(* IEC 61131-3 sources: elevator-digital-twin/codesys, 11 files *)

(* ---- DUT_Types.st ---- *)
(*
    ============================================================================
    DUT_Types.st   —   Asansor Digital Twin / Veri tipleri
    CODESYS 3.5 SP17+  |  Structured Text
    ----------------------------------------------------------------------------
    NOT: Bu dosyadaki her TYPE blogu, CODESYS projesinde AYRI bir DUT nesnesi
         olarak olusturulmalidir (Application > Add Object > DUT).
    NOT: Buradaki sayisal degerler Godot tarafinda scripts/IoMap.gd ve
         scripts/Config.gd icinde birebir ayni tanimlanmistir. Birini
         degistirirseniz digerini de degistirin.
    ============================================================================
*)

// ---------------------------------------------------------------------------
// Ana durum makinesi durumlari  (Godot: IoMap.State)
// ---------------------------------------------------------------------------
TYPE E_LiftState :
(
    LS_INIT         := 0,   // guc geldi, henuz konum bilinmiyor
    LS_HOMING       := 1,   // referans kata inis
    LS_IDLE         := 2,   // bosta, cagri bekliyor
    LS_DOOR_OPENING := 3,
    LS_DOOR_OPEN    := 4,   // bekleme suresi (dwell) sayiyor
    LS_DOOR_CLOSING := 5,
    LS_START        := 6,   // fren cozme + surucu enable
    LS_TRAVEL       := 7,   // nominal hizda seyir
    LS_DECEL        := 8,   // yavaslama rampasi
    LS_LEVEL        := 9,   // kat seviyeleme (surunme hizi)
    LS_ARRIVED      := 10,  // durdu, fren tuttu
    LS_FAULT        := 11,
    LS_FIRE         := 12,  // yangin senaryosu
    LS_INSPECTION   := 13,  // revizyon (kabin ustu kumanda)
    LS_PARK         := 14   // park katina donus
) INT;
END_TYPE

// ---------------------------------------------------------------------------
// Yon  (Godot: IoMap.DIR_*)
// ---------------------------------------------------------------------------
TYPE E_Direction :
(
    DIR_NONE := 0,
    DIR_UP   := 1,
    DIR_DOWN := 2
) INT;
END_TYPE

// ---------------------------------------------------------------------------
// Kapi alt durum makinesi
// ---------------------------------------------------------------------------
TYPE E_DoorState :
(
    DS_CLOSED  := 0,
    DS_OPENING := 1,
    DS_OPEN    := 2,
    DS_CLOSING := 3,
    DS_REOPEN  := 4,   // foto bariyer kesildi, geri ac
    DS_FAULT   := 5
) INT;
END_TYPE

// ---------------------------------------------------------------------------
// Hata kodlari  (Godot: IoMap.FAULT_TEXT)
// ---------------------------------------------------------------------------
TYPE E_Fault :
(
    FLT_NONE          := 0,
    FLT_SAFETY_CHAIN  := 1,   // guvenlik devresi acik
    FLT_DOOR_TIMEOUT  := 2,   // kapi verilen surede kapanmadi/acilmadi
    FLT_TRAVEL_TIMEOUT:= 3,   // kat arasi sure asildi
    FLT_DRIVE         := 4,   // surucu hazir degil / surucu arizasi
    FLT_LIMIT         := 5,   // ucdaki limit switch'e carpildi
    FLT_ENCODER       := 6,   // encoder ile kat sensoru uyusmuyor
    FLT_LOCK_LOST     := 7,   // hareket sirasinda kapi kilidi acildi
    FLT_ESTOP         := 8,   // acil stop butonu
    FLT_BRAKE         := 9,   // fren geri beslemesi kumandayla uyusmuyor
    FLT_OVERSPEED     := 10   // hiz regulatoru devreye girdi
) INT;
END_TYPE

// ---------------------------------------------------------------------------
// Cagri kayit kumesi — dispatcher bu yapinin uzerinde calisir
// ---------------------------------------------------------------------------
TYPE ST_CallSet :
STRUCT
    axUp   : ARRAY[0..15] OF BOOL;   // kat holu YUKARI cagrilari
    axDown : ARRAY[0..15] OF BOOL;   // kat holu ASAGI cagrilari
    axCar  : ARRAY[0..15] OF BOOL;   // kabin ici kat butonlari
END_STRUCT
END_TYPE

// ---------------------------------------------------------------------------
// Sahadan gelen sinyaller  (Godot fizik modeli uretir -> Modbus -> buraya)
// ---------------------------------------------------------------------------
TYPE ST_LiftInputs :
STRUCT
    // Butonlar (momentary)
    stCalls        : ST_CallSet;
    xDoorOpenBtn   : BOOL;
    xDoorCloseBtn  : BOOL;
    xAlarmBtn      : BOOL;
    xFaultReset    : BOOL;

    // Kuyu / kabin sensorleri
    axFloorZone    : ARRAY[0..15] OF BOOL;  // kat seviye (door zone) bayragi
    diPosMM        : DINT;                  // mutlak encoder konumu [mm]
    iActSpeedMMS   : INT;                   // gercek hiz [mm/s]
    iDoorPosPmil   : INT;                   // kapi konumu 0..1000 (0=kapali)
    iLoadKg        : INT;

    // Guvenlik zinciri ve limitler
    xTopLimit      : BOOL;
    xBotLimit      : BOOL;
    xDoorOpenLimit : BOOL;
    xDoorCloseLimit: BOOL;
    xDoorLocked    : BOOL;   // kat kapisi kilit kontagi zinciri
    xBrakeFb       : BOOL;   // fren geri bildirimi
    xSafetyChain   : BOOL;   // TRUE = zincir saglam
    xGovernorOk    : BOOL;   // hiz regulatoru saglam

    // Mod secicileri
    xEStop         : BOOL;
    xOverload      : BOOL;
    xObstruction   : BOOL;   // foto bariyer kesildi
    xFireCall      : BOOL;
    xInspection    : BOOL;
    xInspUp        : BOOL;
    xInspDown      : BOOL;
    xDriveReady    : BOOL;
    xDriveFault    : BOOL;
END_STRUCT
END_TYPE

// ---------------------------------------------------------------------------
// PLC cikislari  (Modbus -> Godot fizik modeli + gorsel)
// ---------------------------------------------------------------------------
TYPE ST_LiftOutputs :
STRUCT
    // Surucu
    xDriveEnable  : BOOL;
    xRunUp        : BOOL;
    xRunDown      : BOOL;
    xBrakeRelease : BOOL;
    xLeveling     : BOOL;
    iSpeedSpMMS   : INT;

    // Kapi
    xDoorOpen     : BOOL;
    xDoorClose    : BOOL;
    xDoorNudge    : BOOL;   // yavas zorlamali kapama

    // Lambalar
    axLampUp      : ARRAY[0..15] OF BOOL;
    axLampDown    : ARRAY[0..15] OF BOOL;
    axLampCar     : ARRAY[0..15] OF BOOL;

    // Gosterge / durum
    iCurrentFloor : INT;
    iTargetFloor  : INT;
    eDirection    : E_Direction;
    eState        : E_LiftState;
    eFault        : E_Fault;
    xMoving       : BOOL;
    xDoorIsOpen   : BOOL;
    xDoorIsClosed : BOOL;
    xOverloadLamp : BOOL;
    xFaultLamp    : BOOL;
    xFireMode     : BOOL;
    xInspMode     : BOOL;
    xOutOfService : BOOL;
    xGong         : BOOL;
    xAlarm        : BOOL;   // alarm zili (kabin alarm butonu)
    xCabinLight   : BOOL;
    iDoorTimerMs  : INT;    // kalan bekleme suresi [ms]
    iHeartbeat    : INT;
END_STRUCT
END_TYPE

(* ---- GVL_Config.st ---- *)
(*
    ============================================================================
    GVL_Config   —   Tesis parametreleri (tek kaynak)
    Application > Add Object > Global Variable List  adiyla: GVL_Config
    ----------------------------------------------------------------------------
    !! Godot tarafindaki karsiligi: godot/scripts/Config.gd
       Iki dosyadaki degerler ayni olmak zorunda, yoksa twin ile gercek PLC
       farkli davranir.
    ============================================================================
*)
VAR_GLOBAL CONSTANT

    // --- Kuyu geometrisi ----------------------------------------------------
    C_FLOOR_COUNT      : INT  := 6;      // 0 = zemin ... 5 = en ust kat
    C_TOP_FLOOR        : INT  := 5;
    C_FLOOR_HEIGHT_MM  : DINT := 3200;   // katlar arasi mesafe
    C_DOOR_ZONE_MM     : DINT := 60;     // kat seviyesi +/- door-zone bolgesi
    C_LEVEL_TOL_MM     : DINT := 8;      // "kata geldi" toleransi
    C_OVERTRAVEL_MM    : DINT := 400;    // ucdaki limit switch mesafesi

    // --- Surus profili ------------------------------------------------------
    C_V_RATED_MMS      : INT  := 1600;   // nominal hiz
    C_V_LEVEL_MMS      : INT  := 150;    // seviyeleme (surunme) hizi
    C_V_INSPECT_MMS    : INT  := 300;    // revizyon hizi
    C_V_OVERSPEED_MMS  : INT  := 1840;   // regulator devreye girme hizi (%115)
    C_DECEL_DIST_MM    : DINT := 2000;   // yavaslamaya baslama mesafesi
                                         // (jerk sinirli surucunun durma
                                         //  mesafesine gore boyutlandirildi)

    // --- Zamanlar -----------------------------------------------------------
    C_T_DOOR_DWELL     : TIME := T#4S;    // kabin cagrisinda kapi acik kalma
    C_T_DOOR_DWELL_HALL: TIME := T#3S;    // sadece hol cagrisinda
    C_T_DOOR_MOVE_MAX  : TIME := T#8S;    // kapi hareket zaman asimi
    C_T_TRAVEL_MAX     : TIME := T#25S;   // kat arasi hareket zaman asimi
    C_T_NUDGE          : TIME := T#15S;   // bu sureden sonra zorlamali kapama
    C_T_GONG           : TIME := T#600MS;
    C_T_PARK           : TIME := T#30S;   // bosta bekleyince park katina don
    C_T_BRAKE          : TIME := T#300MS; // fren cozme/tutma gecikmesi
    C_T_START_DELAY    : TIME := T#200MS; // surucu enable -> hareket
    C_T_ALARM          : TIME := T#2S;    // alarm zili calma suresi
    C_T_BRAKE_FB       : TIME := T#1S;    // fren geri besleme denetimi
    C_T_OVERSPEED      : TIME := T#300MS; // asiri hiz onaylama suresi

    // --- Kat / yuk ----------------------------------------------------------
    C_PARK_FLOOR       : INT  := 0;
    C_FIRE_FLOOR       : INT  := 0;      // yangin tahliye kati
    C_LOAD_FULL_KG     : INT  := 630;
    C_LOAD_OVER_KG     : INT  := 693;    // %110 -> asiri yuk

END_VAR

(* ---- GVL_IO.st ---- *)
(*
    ============================================================================
    GVL_IO   —   Modbus TCP Slave Device register alani
    Application > Add Object > Global Variable List  adiyla: GVL_IO
    ----------------------------------------------------------------------------
    CODESYS "Modbus TCP Slave Device" mantigi:
       Holding Registers  -> PLC girisi  (%IW)  : Godot yazar, PLC okur
       Input Registers    -> PLC cikisi  (%QW)  : PLC yazar, Godot okur

    ONEMLI: Asagidaki %IW0 / %QW0 baslangic adresleri sizin projenizde farkli
    olabilir. Cihaz agacinda "Modbus_TCP_Slave_Device > Modbus TCP Slave Device
    I/O Mapping" sekmesini acip gercek baslangic adresini gorun ve buradaki
    AT ifadelerini ona gore duzeltin.

    Alternatif (AT kullanmak istemezseniz): AT ifadelerini silin, dizileri
    normal degisken birakin ve I/O Mapping sekmesinde her kanali tek tek
    GVL_IO.g_awMbIn[x] / g_awMbOut[x] degiskenine baglayin.
    ============================================================================
*)
VAR_GLOBAL

    // Godot -> PLC  (Holding Registers, master write)
    g_awMbIn  AT %IW0 : ARRAY[0..15] OF WORD;

    // PLC -> Godot  (Input Registers, master read)
    g_awMbOut AT %QW0 : ARRAY[0..15] OF WORD;

    // Uygulama katmani (PRG_ModbusIO tarafindan doldurulur / okunur)
    g_stIn  : ST_LiftInputs;
    g_stOut : ST_LiftOutputs;

    // Baglanti gozetimi
    g_xTwinOnline   : BOOL;        // Godot heartbeat degisiyor mu
    g_iTwinHbLast   : INT;
    g_tTwinLostTime : TIME;

END_VAR

(*
    ============================================================================
    REGISTER HARITASI  (docs/io-map.md ile ayni)
    ----------------------------------------------------------------------------
    Godot -> PLC   g_awMbIn[n]    (Holding Register n)
      0  HALL_UP        bit n = n. kat YUKARI cagri butonu
      1  HALL_DOWN      bit n = n. kat ASAGI cagri butonu
      2  CAR_CALL       bit n = kabin ici n. kat butonu
      3  CMD_BITS       0 kapi-ac btn      1 kapi-kapa btn   2 alarm
                        3 acil stop        4 asiri yuk       5 yangin cagrisi
                        6 revizyon         7 hata reset      8 foto bariyer
                        9 surucu hazir    10 surucu ariza   11 revizyon YUKARI
                       12 revizyon ASAGI
      4  FLOOR_ZONE     bit n = kabin n. katin door-zone bolgesinde
      5  LIMIT_BITS     0 ust limit        1 alt limit       2 kapi acik limit
                        3 kapi kapali lim. 4 kapi kilidi     5 fren geri bes.
                        6 guvenlik zinciri 7 hiz regulatoru
      6  CAR_POS_MM     mutlak konum [mm]  (0..65535)
      7  CAR_SPEED_MMS  gercek hiz [mm/s]
      8  DOOR_POS_PMIL  kapi konumu 0..1000
      9  LOAD_KG        kabin yuku [kg]
     10  TWIN_HB        Godot heartbeat (her cevrim +1)
     11..15  rezerve

    PLC -> Godot   g_awMbOut[n]   (Input Register n)
      0  DRIVE_CMD      0 enable  1 yukari  2 asagi  3 fren-coz  4 seviyeleme
      1  DOOR_CMD       0 ac      1 kapa    2 nudge
      2  LAMP_HALL_UP   bit n
      3  LAMP_HALL_DOWN bit n
      4  LAMP_CAR       bit n
      5  STATUS_BITS    0 hareket  1 kapi acik  2 kapi kapali  3 asiri yuk
                        4 ariza    5 yangin     6 revizyon     7 servis disi
                        8 gong     9 ok-yukari 10 ok-asagi    11 kabin lambasi
                       12 alarm zili
      6  CURRENT_FLOOR
      7  TARGET_FLOOR
      8  DIRECTION      0 yok 1 yukari 2 asagi
      9  SPEED_SP_MMS   hiz referansi [mm/s]
     10  STATE_CODE     E_LiftState
     11  FAULT_CODE     E_Fault
     12  PLC_HB         PLC heartbeat
     13  DOOR_TIMER_MS  kapi bekleme kalan sure [ms]
     14..15  rezerve
    ============================================================================
*)

(* ---- FUN_Bits.st ---- *)
(*
    ============================================================================
    Bit yardimci fonksiyonlari
    Her FUNCTION ayri bir POU olarak eklenmelidir (Add Object > POU > Function).
    ============================================================================
*)

FUNCTION F_GetBit : BOOL
VAR_INPUT
    wVal : WORD;
    iBit : INT;
END_VAR

IF (iBit < 0) OR (iBit > 15) THEN
    F_GetBit := FALSE;
ELSE
    F_GetBit := (wVal AND SHL(WORD#1, INT_TO_BYTE(iBit))) <> 0;
END_IF

END_FUNCTION

FUNCTION F_SetBit : WORD
VAR_INPUT
    wVal : WORD;
    iBit : INT;
    xVal : BOOL;
END_VAR

IF (iBit < 0) OR (iBit > 15) THEN
    F_SetBit := wVal;
ELSIF xVal THEN
    F_SetBit := wVal OR SHL(WORD#1, INT_TO_BYTE(iBit));
ELSE
    F_SetBit := wVal AND (NOT SHL(WORD#1, INT_TO_BYTE(iBit)));
END_IF

END_FUNCTION

(* ---- FB_CallRegistry.st ---- *)
(*
    ============================================================================
    FB_CallRegistry   —   Cagri kaydi (latch) ve lamba surme
    ----------------------------------------------------------------------------
    Butonlar momentary gelir; bu blok cagriyi tutar, servis edilince siler.
    Godot karsiligi: SoftPlc.gd -> class CallRegistry
    ============================================================================
*)
FUNCTION_BLOCK FB_CallRegistry
VAR_INPUT
    stBtn       : ST_CallSet;     // sahadan gelen anlik buton durumu
    xClearAll   : BOOL;           // yangin / revizyon / ariza -> tum cagrilari sil
    xEnable     : BOOL;           // FALSE ise yeni cagri kabul etme
END_VAR
VAR_IN_OUT
    stLatch     : ST_CallSet;     // kalici cagri kaydi (dispatcher ile paylasilir)
END_VAR
VAR_OUTPUT
    xAnyCall    : BOOL;
    iCallCount  : INT;
END_VAR
VAR
    i : INT;
END_VAR

// ---------------------------------------------------------------------------
IF xClearAll THEN
    FOR i := 0 TO 15 DO
        stLatch.axUp[i]   := FALSE;
        stLatch.axDown[i] := FALSE;
        stLatch.axCar[i]  := FALSE;
    END_FOR
    xAnyCall   := FALSE;
    iCallCount := 0;
    RETURN;
END_IF

xAnyCall   := FALSE;
iCallCount := 0;

FOR i := 0 TO C_TOP_FLOOR DO

    // --- yeni cagrilari yakala -------------------------------------------
    IF xEnable THEN
        // en ust katta yukari, en alt katta asagi butonu yoktur
        IF stBtn.axUp[i]   AND (i < C_TOP_FLOOR) THEN stLatch.axUp[i]   := TRUE; END_IF
        IF stBtn.axDown[i] AND (i > 0)           THEN stLatch.axDown[i] := TRUE; END_IF
        IF stBtn.axCar[i]                        THEN stLatch.axCar[i]  := TRUE; END_IF
    END_IF

    // --- sayim -------------------------------------------------------------
    IF stLatch.axUp[i]   THEN iCallCount := iCallCount + 1; END_IF
    IF stLatch.axDown[i] THEN iCallCount := iCallCount + 1; END_IF
    IF stLatch.axCar[i]  THEN iCallCount := iCallCount + 1; END_IF

END_FOR

xAnyCall := (iCallCount > 0);

(*
    ---------------------------------------------------------------------------
    METHOD ServeFloor : Bir katta durulduğunda o kata ait cagrilari siler.
    eDir = hangi yonun cagrisi servis edildi (DIR_NONE ise ikisi de silinir)
    ---------------------------------------------------------------------------
*)
METHOD ServeFloor
VAR_INPUT
    iFloor : INT;
    eDir   : E_Direction;
END_VAR

IF (iFloor < 0) OR (iFloor > C_TOP_FLOOR) THEN RETURN; END_IF

stLatch.axCar[iFloor] := FALSE;

CASE eDir OF
    DIR_UP:
        stLatch.axUp[iFloor] := FALSE;
        // ileride cagri kalmadiysa ters yon cagrisini da al
        IF NOT THIS^.CallAbove(iFloor) THEN
            stLatch.axDown[iFloor] := FALSE;
        END_IF

    DIR_DOWN:
        stLatch.axDown[iFloor] := FALSE;
        IF NOT THIS^.CallBelow(iFloor) THEN
            stLatch.axUp[iFloor] := FALSE;
        END_IF
ELSE
    stLatch.axUp[iFloor]   := FALSE;
    stLatch.axDown[iFloor] := FALSE;
END_CASE

END_METHOD

(*  Verilen katin USTUNDE bekleyen herhangi bir cagri var mi?  *)
METHOD CallAbove : BOOL
VAR_INPUT
    iFloor : INT;
END_VAR
VAR
    k : INT;
END_VAR

CallAbove := FALSE;
FOR k := iFloor + 1 TO C_TOP_FLOOR DO
    IF stLatch.axUp[k] OR stLatch.axDown[k] OR stLatch.axCar[k] THEN
        CallAbove := TRUE;
        RETURN;
    END_IF
END_FOR

END_METHOD

(*  Verilen katin ALTINDA bekleyen herhangi bir cagri var mi?  *)
METHOD CallBelow : BOOL
VAR_INPUT
    iFloor : INT;
END_VAR
VAR
    k : INT;
END_VAR

CallBelow := FALSE;
FOR k := 0 TO iFloor - 1 DO
    IF stLatch.axUp[k] OR stLatch.axDown[k] OR stLatch.axCar[k] THEN
        CallBelow := TRUE;
        RETURN;
    END_IF
END_FOR

END_METHOD

(* ---- FB_Dispatcher.st ---- *)
(*
    ============================================================================
    FB_Dispatcher   —   Hedef kat secimi  (collective control / toplamali kumanda)
    ----------------------------------------------------------------------------
    Kural:
      * Kabin bir yone gidiyorsa o yondeki tum cagrilari sirasiyla toplar.
      * Yonunde is kalmayinca ters yone doner.
      * Bosta ise en yakin cagriya gore yon secer.
    Godot karsiligi: SoftPlc.gd -> class Dispatcher
    ============================================================================
*)
FUNCTION_BLOCK FB_Dispatcher
VAR_INPUT
    iCurrentFloor : INT;
    eCurDir       : E_Direction;   // su anki servis yonu
END_VAR
VAR_IN_OUT
    stLatch : ST_CallSet;
END_VAR
VAR_OUTPUT
    iTarget  : INT := -1;
    eNewDir  : E_Direction := DIR_NONE;
    xHasJob  : BOOL;
END_VAR
VAR
    iBest : INT;
END_VAR

// ---------------------------------------------------------------------------
xHasJob := FALSE;
iTarget := -1;
eNewDir := eCurDir;

// 1) Mevcut yonde devam edilebiliyor mu?
IF eCurDir = DIR_UP THEN
    iBest := THIS^.NearestAbove(iCurrentFloor);
    IF iBest >= 0 THEN
        iTarget := iBest;  eNewDir := DIR_UP;  xHasJob := TRUE;
        RETURN;
    END_IF
    // yukarida is yok -> asagi don
    iBest := THIS^.FarthestBelow(iCurrentFloor);
    IF iBest >= 0 THEN
        iTarget := THIS^.NearestBelow(iCurrentFloor);
        eNewDir := DIR_DOWN;  xHasJob := TRUE;
        RETURN;
    END_IF

ELSIF eCurDir = DIR_DOWN THEN
    iBest := THIS^.NearestBelow(iCurrentFloor);
    IF iBest >= 0 THEN
        iTarget := iBest;  eNewDir := DIR_DOWN;  xHasJob := TRUE;
        RETURN;
    END_IF
    iBest := THIS^.FarthestAbove(iCurrentFloor);
    IF iBest >= 0 THEN
        iTarget := THIS^.NearestAbove(iCurrentFloor);
        eNewDir := DIR_UP;  xHasJob := TRUE;
        RETURN;
    END_IF
END_IF

// 2) Bosta: ayni katta cagri var mi?
IF THIS^.CallAtFloor(iCurrentFloor) THEN
    iTarget := iCurrentFloor;
    eNewDir := DIR_NONE;
    xHasJob := TRUE;
    RETURN;
END_IF

// 3) Bosta: en yakin cagriyi sec
iBest := THIS^.NearestAny(iCurrentFloor);
IF iBest >= 0 THEN
    iTarget := iBest;
    xHasJob := TRUE;
    IF iBest > iCurrentFloor THEN
        eNewDir := DIR_UP;
    ELSIF iBest < iCurrentFloor THEN
        eNewDir := DIR_DOWN;
    ELSE
        eNewDir := DIR_NONE;
    END_IF
ELSE
    eNewDir := DIR_NONE;
END_IF

(*  Gidis yonundeyken bu katta durmali miyiz?  (seyir sirasinda sorulur)  *)
METHOD StopHere : BOOL
VAR_INPUT
    iFloor : INT;
    eDir   : E_Direction;
END_VAR

StopHere := FALSE;
IF (iFloor < 0) OR (iFloor > C_TOP_FLOOR) THEN RETURN; END_IF

// Kabin ici cagri her zaman durdurur
IF stLatch.axCar[iFloor] THEN
    StopHere := TRUE;
    RETURN;
END_IF

CASE eDir OF
    DIR_UP:
        IF stLatch.axUp[iFloor] THEN
            StopHere := TRUE;
        ELSIF stLatch.axDown[iFloor] AND NOT THIS^.AnyAbove(iFloor) THEN
            StopHere := TRUE;   // en ust cagri, ters yon icin de dur
        END_IF

    DIR_DOWN:
        IF stLatch.axDown[iFloor] THEN
            StopHere := TRUE;
        ELSIF stLatch.axUp[iFloor] AND NOT THIS^.AnyBelow(iFloor) THEN
            StopHere := TRUE;
        END_IF
ELSE
    StopHere := THIS^.CallAtFloor(iFloor);
END_CASE

END_METHOD

METHOD CallAtFloor : BOOL
VAR_INPUT
    iFloor : INT;
END_VAR
IF (iFloor < 0) OR (iFloor > C_TOP_FLOOR) THEN
    CallAtFloor := FALSE;
ELSE
    CallAtFloor := stLatch.axUp[iFloor] OR stLatch.axDown[iFloor] OR stLatch.axCar[iFloor];
END_IF
END_METHOD

METHOD AnyAbove : BOOL
VAR_INPUT
    iFloor : INT;
END_VAR
VAR
    k : INT;
END_VAR
AnyAbove := FALSE;
FOR k := iFloor + 1 TO C_TOP_FLOOR DO
    IF THIS^.CallAtFloor(k) THEN AnyAbove := TRUE; RETURN; END_IF
END_FOR
END_METHOD

METHOD AnyBelow : BOOL
VAR_INPUT
    iFloor : INT;
END_VAR
VAR
    k : INT;
END_VAR
AnyBelow := FALSE;
FOR k := 0 TO iFloor - 1 DO
    IF THIS^.CallAtFloor(k) THEN AnyBelow := TRUE; RETURN; END_IF
END_FOR
END_METHOD

METHOD NearestAbove : INT
VAR_INPUT
    iFloor : INT;
END_VAR
VAR
    k : INT;
END_VAR
NearestAbove := -1;
FOR k := iFloor + 1 TO C_TOP_FLOOR DO
    IF THIS^.CallAtFloor(k) THEN NearestAbove := k; RETURN; END_IF
END_FOR
END_METHOD

METHOD NearestBelow : INT
VAR_INPUT
    iFloor : INT;
END_VAR
VAR
    k : INT;
END_VAR
NearestBelow := -1;
FOR k := iFloor - 1 TO 0 BY -1 DO
    IF THIS^.CallAtFloor(k) THEN NearestBelow := k; RETURN; END_IF
END_FOR
END_METHOD

METHOD FarthestAbove : INT
VAR_INPUT
    iFloor : INT;
END_VAR
VAR
    k : INT;
END_VAR
FarthestAbove := -1;
FOR k := C_TOP_FLOOR TO iFloor + 1 BY -1 DO
    IF THIS^.CallAtFloor(k) THEN FarthestAbove := k; RETURN; END_IF
END_FOR
END_METHOD

METHOD FarthestBelow : INT
VAR_INPUT
    iFloor : INT;
END_VAR
VAR
    k : INT;
END_VAR
FarthestBelow := -1;
FOR k := 0 TO iFloor - 1 DO
    IF THIS^.CallAtFloor(k) THEN FarthestBelow := k; RETURN; END_IF
END_FOR
END_METHOD

(*  Yon farketmeksizin en yakin cagri  *)
METHOD NearestAny : INT
VAR_INPUT
    iFloor : INT;
END_VAR
VAR
    d, iUp, iDn : INT;
END_VAR

NearestAny := -1;
iUp := THIS^.NearestAbove(iFloor);
iDn := THIS^.NearestBelow(iFloor);

IF (iUp < 0) AND (iDn < 0) THEN
    RETURN;
ELSIF iUp < 0 THEN
    NearestAny := iDn;
ELSIF iDn < 0 THEN
    NearestAny := iUp;
ELSE
    d := (iUp - iFloor) - (iFloor - iDn);
    IF d <= 0 THEN
        NearestAny := iUp;    // esitlikte yukari onceligi
    ELSE
        NearestAny := iDn;
    END_IF
END_IF

END_METHOD

(* ---- FB_DoorCtrl.st ---- *)
(*
    ============================================================================
    FB_DoorCtrl   —   Kapi alt durum makinesi
    ----------------------------------------------------------------------------
    Kabin kapisi + kat kapisi birlikte surulur (kavrama/coupler mantigi).
    Foto bariyer, kapi-ac butonu ve asiri yuk kapiyi geri actirir.
    C_T_NUDGE suresi asilirsa "nudge" (yavas zorlamali kapama) devreye girer.
    Godot karsiligi: SoftPlc.gd -> class DoorCtrl
    ============================================================================
*)
FUNCTION_BLOCK FB_DoorCtrl
VAR_INPUT
    xEnable       : BOOL;    // FALSE -> kapi motorlari serbest (ariza/estop)
    xReqOpen      : BOOL;    // ust mantik: kapiyi ac ve acik tut
    xReqClose     : BOOL;    // ust mantik: kapiyi kapat (hareket edecegiz)
    xOpenLimit    : BOOL;
    xCloseLimit   : BOOL;
    xObstruction  : BOOL;    // foto bariyer kesildi
    xOpenBtn      : BOOL;
    xCloseBtn     : BOOL;
    xOverload     : BOOL;
    tDwell        : TIME := T#4S;
END_VAR
VAR_OUTPUT
    xOpenOut   : BOOL;
    xCloseOut  : BOOL;
    xNudge     : BOOL;
    xIsOpen    : BOOL;
    xIsClosed  : BOOL;
    xDwellDone : BOOL;       // bekleme suresi doldu, kapanmaya hazir
    xFault     : BOOL;
    eState     : E_DoorState;
    iRemainMs  : INT;
END_VAR
VAR
    tonDwell  : TON;
    tonMove   : TON;         // hareket zaman asimi
    tonNudge  : TON;         // kapida cok bekleme
    tRemain   : TIME;
END_VAR

// ---------------------------------------------------------------------------
// Varsayilan cikislar
xOpenOut   := FALSE;
xCloseOut  := FALSE;
xIsOpen    := xOpenLimit;
xIsClosed  := xCloseLimit;
xDwellDone := FALSE;

IF NOT xEnable THEN
    eState := DS_CLOSED;
    tonDwell(IN := FALSE);
    tonMove(IN := FALSE);
    tonNudge(IN := FALSE);
    xNudge := FALSE;
    iRemainMs := 0;
    RETURN;
END_IF

// ---------------------------------------------------------------------------
CASE eState OF

    // -----------------------------------------------------------------------
    DS_CLOSED:
        tonDwell(IN := FALSE);
        tonNudge(IN := FALSE);
        xNudge := FALSE;
        IF xReqOpen OR xOpenBtn THEN
            eState := DS_OPENING;
        ELSIF NOT xCloseLimit AND xReqClose THEN
            eState := DS_CLOSING;      // tam kapanmamis, tekrar dene
        END_IF

    // -----------------------------------------------------------------------
    DS_OPENING:
        xOpenOut := TRUE;
        tonMove(IN := TRUE, PT := C_T_DOOR_MOVE_MAX);
        IF xOpenLimit THEN
            tonMove(IN := FALSE);
            eState := DS_OPEN;
        ELSIF tonMove.Q THEN
            tonMove(IN := FALSE);
            xFault := TRUE;
            eState := DS_FAULT;
        END_IF

    // -----------------------------------------------------------------------
    DS_OPEN:
        // Bekleme suresi: engel / asiri yuk / ac butonu varken sayac resetlenir
        tonDwell(IN := NOT (xObstruction OR xOverload OR xOpenBtn OR xReqOpen),
                 PT := tDwell);
        tonNudge(IN := TRUE, PT := C_T_NUDGE);
        xNudge := tonNudge.Q;

        tRemain   := tDwell - tonDwell.ET;
        iRemainMs := TIME_TO_INT(tRemain);

        xDwellDone := tonDwell.Q;

        // Kapat butonu bekleme suresini atlatir (engel yoksa)
        IF xCloseBtn AND NOT xObstruction AND NOT xOverload AND NOT xReqOpen THEN
            eState := DS_CLOSING;
            tonDwell(IN := FALSE);
        ELSIF tonDwell.Q AND xReqClose THEN
            eState := DS_CLOSING;
            tonDwell(IN := FALSE);
        ELSIF xNudge AND xReqClose THEN
            eState := DS_CLOSING;      // zorlamali kapama
            tonDwell(IN := FALSE);
        END_IF

    // -----------------------------------------------------------------------
    DS_CLOSING:
        xCloseOut := TRUE;
        tonMove(IN := TRUE, PT := C_T_DOOR_MOVE_MAX);
        iRemainMs := 0;

        // Geri acma sebepleri (nudge modunda foto bariyer yoksayilir,
        // ama ac butonu ve asiri yuk her zaman gecerlidir)
        IF xOpenBtn OR xReqOpen OR xOverload OR (xObstruction AND NOT xNudge) THEN
            tonMove(IN := FALSE);
            eState := DS_REOPEN;
        ELSIF xCloseLimit THEN
            tonMove(IN := FALSE);
            tonNudge(IN := FALSE);
            xNudge := FALSE;
            eState := DS_CLOSED;
        ELSIF tonMove.Q THEN
            tonMove(IN := FALSE);
            xFault := TRUE;
            eState := DS_FAULT;
        END_IF

    // -----------------------------------------------------------------------
    DS_REOPEN:
        xOpenOut := TRUE;
        IF xOpenLimit THEN
            eState := DS_OPEN;
            tonDwell(IN := FALSE);
        END_IF

    // -----------------------------------------------------------------------
    DS_FAULT:
        xOpenOut  := FALSE;
        xCloseOut := FALSE;
        iRemainMs := 0;
        IF NOT xFault THEN                 // disaridan reset edildi
            IF xCloseLimit THEN
                eState := DS_CLOSED;
            ELSE
                eState := DS_OPENING;
            END_IF
        END_IF

END_CASE

(*  Ariza reset (ust mantik cagirir)  *)
METHOD Reset
xFault := FALSE;
END_METHOD

(* ---- FB_LiftCore.st ---- *)
(*
    ============================================================================
    FB_LiftCore   —   ANA DURUM MAKINESI
    ----------------------------------------------------------------------------
    Alt bloklari orkestra eder:
        FB_Safety        guvenlik / ariza
        FB_CallRegistry  cagri latch + lambalar
        FB_Dispatcher    hedef kat secimi
        FB_DoorCtrl      kapi
        FB_Motion        surucu referansi

    Durum akisi (normal):
        INIT -> HOMING -> IDLE -> DOOR_CLOSING -> START -> TRAVEL -> DECEL
             -> LEVEL -> ARRIVED -> DOOR_OPENING -> DOOR_OPEN -> IDLE ...

    Godot karsiligi: SoftPlc.gd -> class LiftCore   (birebir ayni gecisler)
    ============================================================================
*)
FUNCTION_BLOCK FB_LiftCore
VAR_INPUT
    stIn : ST_LiftInputs;
END_VAR
VAR_OUTPUT
    stOut : ST_LiftOutputs;
END_VAR
VAR
    // --- alt bloklar --------------------------------------------------------
    fbSafety : FB_Safety;
    fbCalls  : FB_CallRegistry;
    fbDisp   : FB_Dispatcher;
    fbDoor   : FB_DoorCtrl;
    fbMotion : FB_Motion;

    // --- kalici veri --------------------------------------------------------
    stLatch     : ST_CallSet;
    eState      : E_LiftState := LS_INIT;
    eDir        : E_Direction := DIR_NONE;
    iCurFloor   : INT := 0;
    iTargetFlr  : INT := -1;
    xHomed      : BOOL;

    // --- yardimcilar --------------------------------------------------------
    tonPark     : TON;
    tonGong     : TON;
    tonStart    : TON;
    tonHb       : TON;
    tofAlarm    : TOF;
    xGongArm    : BOOL;
    xFireParked : BOOL;   // tahliye katina varildi (yangin modu mandali)
    xOverspeed  : BOOL;
    xBrakeBad   : BOOL;
    iHb         : INT;
    xZoneMism   : BOOL;
    xDoorReqOpen: BOOL;
    xDoorReqCls : BOOL;
    xClearCalls : BOOL;
    xServeDone  : BOOL;
    i           : INT;
    iZoneFloor  : INT;
    tDwellUse   : TIME;
END_VAR

// ===========================================================================
// 1) GUVENLIK
// ---------------------------------------------------------------------------
// Regulator (asiri hiz) ve fren geri besleme denetimi: her ikisi de sahadan
// gelen olcumu kumanda ile karsilastirir.
// ===========================================================================
xOverspeed := fbSafety.OverspeedTrip(stIn.iActSpeedMMS);
xBrakeBad  := fbMotion.BrakeMismatch(stOut.xBrakeRelease, stIn.xBrakeFb);

fbSafety(
    xSafetyChain   := stIn.xSafetyChain,
    xGovernorOk    := stIn.xGovernorOk,
    xEStop         := stIn.xEStop,
    xDriveReady    := stIn.xDriveReady,
    xDriveFault    := stIn.xDriveFault,
    xTopLimit      := stIn.xTopLimit,
    xBotLimit      := stIn.xBotLimit,
    xDoorLocked    := stIn.xDoorLocked,
    xMoving        := stOut.xMoving,
    xDoorTimeout   := fbDoor.xFault,
    xTravelTimeout := fbMotion.xTimeout,
    xZoneMismatch  := xZoneMism,
    xOverspeed     := xOverspeed,
    xBrakeMismatch := xBrakeBad,
    xReset         := stIn.xFaultReset
);

// ===========================================================================
// 2) KONUM / KAT TAKIBI
// ===========================================================================
iCurFloor := fbMotion.FloorFromPos(stIn.diPosMM);

// Kat sensoru ile encoder tutarlilik kontrolu (sadece door-zone icinde)
iZoneFloor := -1;
FOR i := 0 TO C_TOP_FLOOR DO
    IF stIn.axFloorZone[i] THEN iZoneFloor := i; END_IF
END_FOR
xZoneMism := (iZoneFloor >= 0) AND (iZoneFloor <> iCurFloor);

// ===========================================================================
// 3) CAGRI KAYDI
// ===========================================================================
xClearCalls := stIn.xFireCall OR stIn.xInspection OR fbSafety.xFault;

fbCalls(
    stBtn     := stIn.stCalls,
    xClearAll := xClearCalls,
    xEnable   := NOT stIn.xInspection AND NOT fbSafety.xFault AND NOT stIn.xFireCall,
    stLatch   := stLatch
);

// ===========================================================================
// 4) HEDEF SECIMI
// ===========================================================================
fbDisp(
    iCurrentFloor := iCurFloor,
    eCurDir       := eDir,
    stLatch       := stLatch
);

// ===========================================================================
// 5) ANA DURUM MAKINESI
// ===========================================================================
xDoorReqOpen := FALSE;
xDoorReqCls  := FALSE;
xServeDone   := FALSE;

// --- global oncelikli gecisler ---------------------------------------------
IF fbSafety.xFault AND (eState <> LS_FAULT) THEN
    eState := LS_FAULT;
ELSIF stIn.xInspection AND (eState <> LS_INSPECTION) AND NOT fbSafety.xFault THEN
    eState := LS_INSPECTION;
ELSIF stIn.xFireCall AND (eState <> LS_FIRE) AND NOT fbSafety.xFault
      AND NOT stIn.xInspection THEN
    eState := LS_FIRE;
END_IF

CASE eState OF

    // -----------------------------------------------------------------------
    LS_INIT:
        eDir       := DIR_NONE;
        iTargetFlr := -1;
        IF fbSafety.xRunAllow THEN
            IF stIn.axFloorZone[iCurFloor] THEN
                xHomed := TRUE;
                eState := LS_IDLE;
            ELSE
                eState := LS_HOMING;
            END_IF
        END_IF

    // -----------------------------------------------------------------------
    // Konum bilinmiyor: en yakin kata surunme hiziyla git
    LS_HOMING:
        xDoorReqCls := TRUE;
        IF fbDoor.xIsClosed AND stIn.xDoorLocked THEN
            iTargetFlr := iCurFloor;
            IF fbMotion.xAtTarget THEN
                xHomed := TRUE;
                eState := LS_ARRIVED;
            END_IF
        END_IF

    // -----------------------------------------------------------------------
    LS_IDLE:
        iTargetFlr := -1;
        tonPark(IN := NOT fbCalls.xAnyCall, PT := C_T_PARK);

        IF fbDisp.xHasJob THEN
            tonPark(IN := FALSE);
            IF fbDisp.iTarget = iCurFloor THEN
                // ayni katta cagri -> kapiyi ac
                eDir       := fbDisp.eNewDir;
                iTargetFlr := iCurFloor;
                xServeDone := TRUE;
                eState     := LS_DOOR_OPENING;
            ELSE
                eDir       := fbDisp.eNewDir;
                iTargetFlr := fbDisp.iTarget;
                fbMotion.ResetTimeout();
                eState     := LS_DOOR_CLOSING;
            END_IF

        ELSIF tonPark.Q AND (iCurFloor <> C_PARK_FLOOR) THEN
            tonPark(IN := FALSE);
            iTargetFlr := C_PARK_FLOOR;
            IF iCurFloor > C_PARK_FLOOR THEN eDir := DIR_DOWN; ELSE eDir := DIR_UP; END_IF
            fbMotion.ResetTimeout();
            eState := LS_PARK;
        END_IF

    // -----------------------------------------------------------------------
    LS_DOOR_CLOSING:
        xDoorReqCls := TRUE;
        // Asiri yuk KALKISI engeller (seyir halindeki kabini durdurmaz).
        IF fbDoor.xIsClosed AND stIn.xDoorLocked AND NOT stIn.xOverload THEN
            tonStart(IN := TRUE, PT := C_T_START_DELAY);
            IF tonStart.Q THEN
                tonStart(IN := FALSE);
                eState := LS_START;
            END_IF
        ELSE
            tonStart(IN := FALSE);
        END_IF
        // kapanma sirasinda yeni bir cagri ayni kattan gelirse geri ac
        IF stLatch.axCar[iCurFloor] OR stIn.xDoorOpenBtn THEN
            eState := LS_DOOR_OPENING;
        END_IF

    // -----------------------------------------------------------------------
    LS_START:
        xDoorReqCls := TRUE;
        IF fbMotion.xBrakeRelease AND (fbMotion.iSpeedSp > 0) THEN
            eState := LS_TRAVEL;
        END_IF
        IF fbMotion.xAtTarget THEN
            eState := LS_ARRIVED;
        END_IF

    // -----------------------------------------------------------------------
    LS_TRAVEL:
        xDoorReqCls := TRUE;

        // Yol uzerindeki kata ugrama karari (door-zone'a girmeden once verilir)
        IF (iZoneFloor >= 0) AND (iZoneFloor <> iTargetFlr) THEN
            IF fbDisp.StopHere(iZoneFloor, eDir) THEN
                iTargetFlr := iZoneFloor;
                fbMotion.ResetTimeout();
            END_IF
        END_IF

        IF fbMotion.xLeveling THEN
            eState := LS_LEVEL;
        ELSIF ABS(fbMotion.diErrMM) < C_DECEL_DIST_MM THEN
            eState := LS_DECEL;
        END_IF

    // -----------------------------------------------------------------------
    LS_DECEL:
        xDoorReqCls := TRUE;
        IF fbMotion.xLeveling THEN
            eState := LS_LEVEL;
        END_IF

    // -----------------------------------------------------------------------
    LS_LEVEL:
        xDoorReqCls := TRUE;
        IF fbMotion.xAtTarget THEN
            eState := LS_ARRIVED;
        END_IF

    // -----------------------------------------------------------------------
    LS_ARRIVED:
        iTargetFlr := -1;
        xServeDone := TRUE;
        // Gong burada KURULUR; calma suresi durum degisiminden bagimsiz
        // olarak asagida sayilir (LS_ARRIVED yalnizca tek tarama surer).
        xGongArm := TRUE;
        tonGong(IN := FALSE);

        // Bu kat icin cagrilari sil ve kapiyi ac
        eState := LS_DOOR_OPENING;

    // -----------------------------------------------------------------------
    LS_DOOR_OPENING:
        xDoorReqOpen := TRUE;
        IF fbDoor.eState = DS_OPEN THEN
            eState := LS_DOOR_OPEN;
        END_IF

    // -----------------------------------------------------------------------
    LS_DOOR_OPEN:
        // Yeni is varsa kapanmaya izin ver
        xDoorReqCls := fbDisp.xHasJob OR fbDoor.xDwellDone;
        IF fbDoor.eState = DS_CLOSED THEN
            eState := LS_IDLE;
            eDir   := fbDisp.eNewDir;
        END_IF

    // -----------------------------------------------------------------------
    LS_PARK:
        xDoorReqCls := TRUE;
        IF fbDisp.xHasJob THEN
            eDir       := fbDisp.eNewDir;
            iTargetFlr := fbDisp.iTarget;
            fbMotion.ResetTimeout();
            eState     := LS_DOOR_CLOSING;
        ELSIF fbMotion.xAtTarget THEN
            eDir   := DIR_NONE;
            eState := LS_IDLE;
        END_IF

    // -----------------------------------------------------------------------
    // Yangin senaryosu: tum cagrilar silinir, tahliye katina inilir,
    // kapi acilir ve acik kalir.
    LS_FIRE:
        (* Tahliye katina varis MANDALLANIR. Aksi halde kapi acilinca hareket
           blogu devre disi kalir, xAtTarget duser ve kumanda kapiyi yeniden
           kapatmaya calisir (ac-kapa dongusu olusur). *)
        IF NOT xFireParked THEN
            eDir        := DIR_DOWN;
            iTargetFlr  := C_FIRE_FLOOR;
            xDoorReqCls := TRUE;
            IF (iCurFloor = C_FIRE_FLOOR) AND fbMotion.xAtTarget THEN
                xFireParked := TRUE;
            END_IF
        ELSE
            (* tahliye katinda park: surucu serbest, kapi acik kalir *)
            iTargetFlr   := -1;
            eDir         := DIR_NONE;
            xDoorReqOpen := TRUE;
        END_IF

        IF NOT stIn.xFireCall THEN
            xFireParked := FALSE;
            eState := LS_IDLE;
        END_IF

    // -----------------------------------------------------------------------
    LS_INSPECTION:
        iTargetFlr := -1;
        eDir       := DIR_NONE;
        IF NOT stIn.xInspection THEN
            eState := LS_INIT;
        END_IF

    // -----------------------------------------------------------------------
    LS_FAULT:
        iTargetFlr := -1;
        eDir       := DIR_NONE;
        // kabin door-zone icindeyse kapiyi ac (yolcu tahliyesi)
        xDoorReqOpen := (iZoneFloor >= 0);
        IF NOT fbSafety.xFault THEN
            fbDoor.Reset();
            fbMotion.ResetTimeout();
            eState := LS_INIT;
        END_IF

END_CASE

// --- kata varinca cagrilari sil --------------------------------------------
IF xServeDone THEN
    fbCalls.ServeFloor(iCurFloor, eDir);
END_IF

// ===========================================================================
// 5b) GONG VE ALARM ZILI
// ===========================================================================
// Gong LS_ARRIVED'de kurulur, C_T_GONG boyunca calar (durumdan bagimsiz).
IF xGongArm THEN
    tonGong(IN := TRUE, PT := C_T_GONG);
    stOut.xGong := NOT tonGong.Q;
    IF tonGong.Q THEN
        xGongArm := FALSE;
    END_IF
ELSE
    stOut.xGong := FALSE;
END_IF

// Alarm butonu anlik (momentary) gelir; zil basildiktan sonra C_T_ALARM
// suresince calmaya devam eder (TOF = kapanma gecikmesi).
tofAlarm(IN := stIn.xAlarmBtn, PT := C_T_ALARM);
stOut.xAlarm := tofAlarm.Q;

// ===========================================================================
// 6) KAPI
// ===========================================================================
IF stLatch.axCar[iCurFloor] OR (eDir = DIR_NONE) THEN
    tDwellUse := C_T_DOOR_DWELL;
ELSE
    tDwellUse := C_T_DOOR_DWELL_HALL;
END_IF

fbDoor(
    xEnable      := NOT stIn.xEStop AND stIn.xSafetyChain,
    xReqOpen     := xDoorReqOpen,
    xReqClose    := xDoorReqCls,
    xOpenLimit   := stIn.xDoorOpenLimit,
    xCloseLimit  := stIn.xDoorCloseLimit,
    xObstruction := stIn.xObstruction,
    xOpenBtn     := stIn.xDoorOpenBtn,
    xCloseBtn    := stIn.xDoorCloseBtn,
    xOverload    := stIn.xOverload,
    tDwell       := tDwellUse
);

// ===========================================================================
// 7) HAREKET
// ===========================================================================
(*
    Asiri yuk burada YOK: yuk sinyali kalkis kilididir (LS_DOOR_CLOSING),
    seyir halindeki kabini aniden durdurmamalidir.
*)
fbMotion(
    xEnable      := fbSafety.xRunAllow
                    AND fbDoor.xIsClosed
                    AND stIn.xDoorLocked
                    AND xHomed,
    iTargetFloor := iTargetFlr,
    diPosMM      := stIn.diPosMM,
    xTopLimit    := stIn.xTopLimit,
    xBotLimit    := stIn.xBotLimit,
    xInspection  := stIn.xInspection,
    xInspUp      := stIn.xInspUp,
    xInspDown    := stIn.xInspDown
);

// ===========================================================================
// 8) CIKISLAR
// ===========================================================================
stOut.xDriveEnable  := fbMotion.xDriveEnable;
stOut.xRunUp        := fbMotion.xRunUp;
stOut.xRunDown      := fbMotion.xRunDown;
stOut.xBrakeRelease := fbMotion.xBrakeRelease;
stOut.xLeveling     := fbMotion.xLeveling;
stOut.iSpeedSpMMS   := fbMotion.iSpeedSp;

stOut.xDoorOpen     := fbDoor.xOpenOut;
stOut.xDoorClose    := fbDoor.xCloseOut;
stOut.xDoorNudge    := fbDoor.xNudge;
stOut.xDoorIsOpen   := fbDoor.xIsOpen;
stOut.xDoorIsClosed := fbDoor.xIsClosed;
stOut.iDoorTimerMs  := fbDoor.iRemainMs;

FOR i := 0 TO 15 DO
    stOut.axLampUp[i]   := stLatch.axUp[i];
    stOut.axLampDown[i] := stLatch.axDown[i];
    stOut.axLampCar[i]  := stLatch.axCar[i];
END_FOR

stOut.iCurrentFloor := iCurFloor;
stOut.iTargetFloor  := iTargetFlr;
stOut.eDirection    := eDir;
stOut.eState        := eState;
stOut.eFault        := fbSafety.eFault;
stOut.xMoving       := fbMotion.xRunUp OR fbMotion.xRunDown;
stOut.xOverloadLamp := stIn.xOverload;
stOut.xFaultLamp    := fbSafety.xFault;
stOut.xFireMode     := (eState = LS_FIRE);
stOut.xInspMode     := (eState = LS_INSPECTION);
stOut.xOutOfService := fbSafety.xFault OR (eState = LS_INSPECTION) OR (eState = LS_FIRE);
stOut.xCabinLight   := NOT fbSafety.xFault OR (fbSafety.eFault <> FLT_SAFETY_CHAIN);

// Heartbeat: 100 ms'de bir artar
tonHb(IN := NOT tonHb.Q, PT := T#100MS);
IF tonHb.Q THEN
    iHb := iHb + 1;
    IF iHb > 32000 THEN iHb := 0; END_IF
END_IF
stOut.iHeartbeat := iHb;

(* ---- FB_Motion.st ---- *)
(*
    ============================================================================
    FB_Motion   —   Hareket / hiz profili / kat takibi
    ----------------------------------------------------------------------------
    Surucu (VVVF) referansi uretir:  yon + hiz setpoint + fren.
    Profil:
        |hata| >= C_DECEL_DIST_MM        -> nominal hiz
        C_DOOR_ZONE_MM < |hata| < decel  -> lineer yavaslama rampasi
        |hata| <= C_DOOR_ZONE_MM         -> seviyeleme (surunme) hizi
        |hata| <= C_LEVEL_TOL_MM         -> dur, fren tut
    Godot karsiligi: SoftPlc.gd -> class Motion
    ============================================================================
*)
FUNCTION_BLOCK FB_Motion
VAR_INPUT
    xEnable      : BOOL;      // hareket izni (kapi kilitli + guvenlik ok)
    iTargetFloor : INT := -1;
    diPosMM      : DINT;      // encoder mutlak konum
    xTopLimit    : BOOL;
    xBotLimit    : BOOL;
    xInspection  : BOOL;
    xInspUp      : BOOL;
    xInspDown    : BOOL;
END_VAR
VAR_OUTPUT
    xDriveEnable  : BOOL;
    xRunUp        : BOOL;
    xRunDown      : BOOL;
    xBrakeRelease : BOOL;
    xLeveling     : BOOL;
    iSpeedSp      : INT;
    eDir          : E_Direction;
    xAtTarget     : BOOL;
    xTimeout      : BOOL;
    diErrMM       : DINT;
END_VAR
VAR
    diTargetMM : DINT;
    diAbsErr   : DINT;
    tonTravel  : TON;
    tonBrakeFb : TON;
    tonBrake   : TON;
    xMoveReq   : BOOL;
END_VAR

// ---------------------------------------------------------------------------
// Revizyon modu: hedef yok, sadece butona basildigi surece surunme hizinda
// ---------------------------------------------------------------------------
IF xInspection THEN
    xAtTarget := FALSE;
    tonTravel(IN := FALSE);
    xTimeout  := FALSE;

    IF xEnable AND xInspUp AND NOT xInspDown AND NOT xTopLimit THEN
        xDriveEnable := TRUE; xBrakeRelease := TRUE;
        xRunUp := TRUE;  xRunDown := FALSE;
        iSpeedSp := C_V_INSPECT_MMS;  eDir := DIR_UP;
    ELSIF xEnable AND xInspDown AND NOT xInspUp AND NOT xBotLimit THEN
        xDriveEnable := TRUE; xBrakeRelease := TRUE;
        xRunUp := FALSE; xRunDown := TRUE;
        iSpeedSp := C_V_INSPECT_MMS;  eDir := DIR_DOWN;
    ELSE
        xDriveEnable := FALSE; xBrakeRelease := FALSE;
        xRunUp := FALSE; xRunDown := FALSE;
        iSpeedSp := 0;  eDir := DIR_NONE;
    END_IF
    xLeveling := TRUE;
    RETURN;
END_IF

// ---------------------------------------------------------------------------
// Normal mod
// ---------------------------------------------------------------------------
IF (iTargetFloor < 0) OR (iTargetFloor > C_TOP_FLOOR) OR NOT xEnable THEN
    xDriveEnable  := FALSE;
    xRunUp        := FALSE;
    xRunDown      := FALSE;
    xBrakeRelease := FALSE;
    xLeveling     := FALSE;
    iSpeedSp      := 0;
    eDir          := DIR_NONE;
    xAtTarget     := FALSE;
    (* Zamanlayici ile birlikte CIKIS BAYRAGI da temizlenmelidir; aksi halde
       bir kez olusan zaman asimi kalici kalir ve ariza reset edilemez. *)
    tonTravel(IN := FALSE);
    xTimeout      := FALSE;
    RETURN;
END_IF

diTargetMM := INT_TO_DINT(iTargetFloor) * C_FLOOR_HEIGHT_MM;
diErrMM    := diTargetMM - diPosMM;
diAbsErr   := ABS(diErrMM);

// --- hedefe varildi mi? ----------------------------------------------------
IF diAbsErr <= C_LEVEL_TOL_MM THEN
    xAtTarget     := TRUE;
    xMoveReq      := FALSE;
    xRunUp        := FALSE;
    xRunDown      := FALSE;
    iSpeedSp      := 0;
    eDir          := DIR_NONE;
    xLeveling     := FALSE;
    tonTravel(IN := FALSE);

    // fren tutma gecikmesi sonrasi surucuyu birak
    tonBrake(IN := TRUE, PT := C_T_BRAKE);
    xBrakeRelease := NOT tonBrake.Q;
    xDriveEnable  := NOT tonBrake.Q;
    RETURN;
END_IF

xAtTarget := FALSE;
tonBrake(IN := FALSE);

// --- ucdaki limitler -------------------------------------------------------
IF (diErrMM > 0) AND xTopLimit THEN
    xDriveEnable := FALSE; xRunUp := FALSE; xRunDown := FALSE;
    iSpeedSp := 0; xBrakeRelease := FALSE; eDir := DIR_NONE;
    RETURN;
END_IF
IF (diErrMM < 0) AND xBotLimit THEN
    xDriveEnable := FALSE; xRunUp := FALSE; xRunDown := FALSE;
    iSpeedSp := 0; xBrakeRelease := FALSE; eDir := DIR_NONE;
    RETURN;
END_IF

// --- hiz profili -----------------------------------------------------------
IF diAbsErr <= C_DOOR_ZONE_MM THEN
    iSpeedSp  := C_V_LEVEL_MMS;
    xLeveling := TRUE;
ELSIF diAbsErr >= C_DECEL_DIST_MM THEN
    iSpeedSp  := C_V_RATED_MMS;
    xLeveling := FALSE;
ELSE
    // Lineer rampa:  door-zone kenarinda C_V_LEVEL, decel mesafesinde C_V_RATED
    iSpeedSp := C_V_LEVEL_MMS
              + DINT_TO_INT( ((diAbsErr - C_DOOR_ZONE_MM)
                            * INT_TO_DINT(C_V_RATED_MMS - C_V_LEVEL_MMS))
                            / (C_DECEL_DIST_MM - C_DOOR_ZONE_MM) );
    xLeveling := FALSE;
END_IF

// --- yon ve surucu ---------------------------------------------------------
xDriveEnable  := TRUE;
xBrakeRelease := TRUE;

IF diErrMM > 0 THEN
    xRunUp := TRUE;  xRunDown := FALSE;  eDir := DIR_UP;
ELSE
    xRunUp := FALSE; xRunDown := TRUE;   eDir := DIR_DOWN;
END_IF

// --- hareket zaman asimi ---------------------------------------------------
tonTravel(IN := TRUE, PT := C_T_TRAVEL_MAX);
xTimeout := tonTravel.Q;

(*  Yeni hedef verildiginde zaman asimi sayacini sifirla  *)
METHOD ResetTimeout
tonTravel(IN := FALSE);
xTimeout := FALSE;
END_METHOD

(*  Encoder konumundan kat numarasi (en yakin kat)  *)
METHOD FloorFromPos : INT
VAR_INPUT
    diPos : DINT;
END_VAR
VAR
    i : INT;
END_VAR

FloorFromPos := 0;
FOR i := 0 TO C_TOP_FLOOR DO
    IF ABS(diPos - (INT_TO_DINT(i) * C_FLOOR_HEIGHT_MM)) <= (C_FLOOR_HEIGHT_MM / 2) THEN
        FloorFromPos := i;
        RETURN;
    END_IF
END_FOR

IF diPos > (INT_TO_DINT(C_TOP_FLOOR) * C_FLOOR_HEIGHT_MM) THEN
    FloorFromPos := C_TOP_FLOOR;
END_IF

END_METHOD

(*
    Fren geri beslemesi denetimi: kumanda ile saha uyusmali.
    xBrakeCmd = fren coz komutu, xBrakeFb = fren gercekten cozuldu sinyali.
    Uyusmazlik C_T_BRAKE_FB suresince surerse TRUE doner.
    Godot karsiligi: SoftPlc.gd -> Motion.brake_mismatch()
*)
METHOD BrakeMismatch : BOOL
VAR_INPUT
    xBrakeCmd : BOOL;
    xBrakeFb  : BOOL;
END_VAR

tonBrakeFb(IN := (xBrakeCmd <> xBrakeFb), PT := C_T_BRAKE_FB);
BrakeMismatch := tonBrakeFb.Q;

END_METHOD

(* ---- FB_Safety.st ---- *)
(*
    ============================================================================
    FB_Safety   —   Guvenlik denetimi ve ariza yonetimi
    ----------------------------------------------------------------------------
    Onceligi en yuksek olan hata kodu cikar. Ariza kalicidir; reset butonu ile
    (ve hata sebebi ortadan kalkmissa) silinir.
    Godot karsiligi: SoftPlc.gd -> class Safety
    ============================================================================
*)
FUNCTION_BLOCK FB_Safety
VAR_INPUT
    xSafetyChain  : BOOL;   // TRUE = saglam
    xGovernorOk   : BOOL;
    xEStop        : BOOL;
    xDriveReady   : BOOL;
    xDriveFault   : BOOL;
    xTopLimit     : BOOL;
    xBotLimit     : BOOL;
    xDoorLocked   : BOOL;
    xMoving       : BOOL;
    xDoorTimeout  : BOOL;
    xTravelTimeout: BOOL;
    xZoneMismatch : BOOL;   // encoder ile kat sensoru uyusmuyor
    xOverspeed    : BOOL;   // hiz regulatoru devreye girdi
    xBrakeMismatch: BOOL;   // fren geri beslemesi kumandayla uyusmuyor
    xReset        : BOOL;
END_VAR
VAR_OUTPUT
    eFault    : E_Fault;
    xFault    : BOOL;
    xRunAllow : BOOL;       // hareket izni
END_VAR
VAR
    xResetEdge : R_TRIG;
    tonOverspd : TON;
END_VAR

// ---------------------------------------------------------------------------
xResetEdge(CLK := xReset);

// --- Ariza tespiti (oncelik sirasiyla) -------------------------------------
IF eFault = FLT_NONE THEN

    IF xEStop THEN
        eFault := FLT_ESTOP;

    ELSIF NOT xSafetyChain OR NOT xGovernorOk THEN
        eFault := FLT_SAFETY_CHAIN;

    ELSIF xOverspeed THEN
        eFault := FLT_OVERSPEED;

    ELSIF xDriveFault OR NOT xDriveReady THEN
        eFault := FLT_DRIVE;

    ELSIF xBrakeMismatch THEN
        eFault := FLT_BRAKE;

    ELSIF xTopLimit OR xBotLimit THEN
        eFault := FLT_LIMIT;

    ELSIF xMoving AND NOT xDoorLocked THEN
        eFault := FLT_LOCK_LOST;       // hareket halinde kilit acildi

    ELSIF xTravelTimeout THEN
        eFault := FLT_TRAVEL_TIMEOUT;

    ELSIF xDoorTimeout THEN
        eFault := FLT_DOOR_TIMEOUT;

    ELSIF xZoneMismatch THEN
        eFault := FLT_ENCODER;
    END_IF

END_IF

// --- Reset ------------------------------------------------------------------
IF xResetEdge.Q THEN
    // sebep hala duruyorsa reset kabul edilmez
    IF NOT xEStop
       AND xSafetyChain AND xGovernorOk
       AND xDriveReady AND NOT xDriveFault
       AND NOT xTopLimit AND NOT xBotLimit THEN
        eFault := FLT_NONE;
    END_IF
END_IF

xFault    := (eFault <> FLT_NONE);

xRunAllow := NOT xFault
             AND xSafetyChain AND xGovernorOk
             AND xDriveReady AND NOT xDriveFault
             AND NOT xEStop;

(*
    Regulator islevi: gercek hiz anma hizinin %115'ini (C_V_OVERSPEED_MMS)
    C_T_OVERSPEED suresince asarsa devreye girer.
    Godot karsiligi: SoftPlc.gd -> Safety.overspeed_trip()
*)
METHOD OverspeedTrip : BOOL
VAR_INPUT
    iActSpeedMMS : INT;
END_VAR

tonOverspd(IN := (iActSpeedMMS > C_V_OVERSPEED_MMS), PT := C_T_OVERSPEED);
OverspeedTrip := tonOverspd.Q;

END_METHOD

(* ---- PLC_PRG.st ---- *)
(*
    ============================================================================
    PLC_PRG   —   Ana program (Task: 10 ms cyclic onerilir)
    ----------------------------------------------------------------------------
    Akis:
        1) Modbus Holding Register'lari -> ST_LiftInputs        (Godot -> PLC)
        2) FB_LiftCore                                          (kontrol mantigi)
        3) ST_LiftOutputs -> Modbus Input Register'lari          (PLC -> Godot)
        4) Twin baglanti gozetimi (heartbeat)

    Register haritasi icin GVL_IO.st basligina veya docs/io-map.md dosyasina bakin.
    ============================================================================
*)
PROGRAM PLC_PRG
VAR
    fbLift  : FB_LiftCore;

    i       : INT;
    wTmp    : WORD;
    wCmd    : WORD;
    wLim    : WORD;

    // Twin (Godot) baglanti gozetimi
    tonTwinLost : TON;
    iHbPrev     : INT;

    // Manuel test bayraklari (CODESYS izleme penceresinden zorlanabilir)
    xForceOffline : BOOL;
END_VAR

// ===========================================================================
// 1) GIRISLER:  Modbus Holding Registers -> ST_LiftInputs
// ===========================================================================
wCmd := GVL_IO.g_awMbIn[3];
wLim := GVL_IO.g_awMbIn[5];

FOR i := 0 TO 15 DO
    GVL_IO.g_stIn.stCalls.axUp[i]   := F_GetBit(GVL_IO.g_awMbIn[0], i);
    GVL_IO.g_stIn.stCalls.axDown[i] := F_GetBit(GVL_IO.g_awMbIn[1], i);
    GVL_IO.g_stIn.stCalls.axCar[i]  := F_GetBit(GVL_IO.g_awMbIn[2], i);
    GVL_IO.g_stIn.axFloorZone[i]    := F_GetBit(GVL_IO.g_awMbIn[4], i);
END_FOR

// CMD_BITS
GVL_IO.g_stIn.xDoorOpenBtn  := F_GetBit(wCmd,  0);
GVL_IO.g_stIn.xDoorCloseBtn := F_GetBit(wCmd,  1);
GVL_IO.g_stIn.xAlarmBtn     := F_GetBit(wCmd,  2);
GVL_IO.g_stIn.xEStop        := F_GetBit(wCmd,  3);
GVL_IO.g_stIn.xOverload     := F_GetBit(wCmd,  4);
GVL_IO.g_stIn.xFireCall     := F_GetBit(wCmd,  5);
GVL_IO.g_stIn.xInspection   := F_GetBit(wCmd,  6);
GVL_IO.g_stIn.xFaultReset   := F_GetBit(wCmd,  7);
GVL_IO.g_stIn.xObstruction  := F_GetBit(wCmd,  8);
GVL_IO.g_stIn.xDriveReady   := F_GetBit(wCmd,  9);
GVL_IO.g_stIn.xDriveFault   := F_GetBit(wCmd, 10);
GVL_IO.g_stIn.xInspUp       := F_GetBit(wCmd, 11);
GVL_IO.g_stIn.xInspDown     := F_GetBit(wCmd, 12);

// LIMIT_BITS
GVL_IO.g_stIn.xTopLimit       := F_GetBit(wLim, 0);
GVL_IO.g_stIn.xBotLimit       := F_GetBit(wLim, 1);
GVL_IO.g_stIn.xDoorOpenLimit  := F_GetBit(wLim, 2);
GVL_IO.g_stIn.xDoorCloseLimit := F_GetBit(wLim, 3);
GVL_IO.g_stIn.xDoorLocked     := F_GetBit(wLim, 4);
GVL_IO.g_stIn.xBrakeFb        := F_GetBit(wLim, 5);
GVL_IO.g_stIn.xSafetyChain    := F_GetBit(wLim, 6);
GVL_IO.g_stIn.xGovernorOk     := F_GetBit(wLim, 7);

// Analog degerler
GVL_IO.g_stIn.diPosMM      := WORD_TO_DINT(GVL_IO.g_awMbIn[6]);
GVL_IO.g_stIn.iActSpeedMMS := WORD_TO_INT(GVL_IO.g_awMbIn[7]);
GVL_IO.g_stIn.iDoorPosPmil := WORD_TO_INT(GVL_IO.g_awMbIn[8]);
GVL_IO.g_stIn.iLoadKg      := WORD_TO_INT(GVL_IO.g_awMbIn[9]);

// ---------------------------------------------------------------------------
// Twin baglanti gozetimi: heartbeat 2 s degismezse simulasyon kopmustur.
// Bu durumda guvenlik zinciri "acik" sayilir; asansor hareket etmez.
// ---------------------------------------------------------------------------
IF WORD_TO_INT(GVL_IO.g_awMbIn[10]) <> iHbPrev THEN
    iHbPrev := WORD_TO_INT(GVL_IO.g_awMbIn[10]);
    tonTwinLost(IN := FALSE);
    GVL_IO.g_xTwinOnline := TRUE;
END_IF
tonTwinLost(IN := TRUE, PT := T#2S);
IF tonTwinLost.Q OR xForceOffline THEN
    GVL_IO.g_xTwinOnline := FALSE;
END_IF

IF NOT GVL_IO.g_xTwinOnline THEN
    GVL_IO.g_stIn.xSafetyChain := FALSE;
END_IF

// ===========================================================================
// 2) KONTROL MANTIGI
// ===========================================================================
fbLift(stIn := GVL_IO.g_stIn);
GVL_IO.g_stOut := fbLift.stOut;

// ===========================================================================
// 3) CIKISLAR:  ST_LiftOutputs -> Modbus Input Registers
// ===========================================================================

// DRIVE_CMD
wTmp := 0;
wTmp := F_SetBit(wTmp, 0, GVL_IO.g_stOut.xDriveEnable);
wTmp := F_SetBit(wTmp, 1, GVL_IO.g_stOut.xRunUp);
wTmp := F_SetBit(wTmp, 2, GVL_IO.g_stOut.xRunDown);
wTmp := F_SetBit(wTmp, 3, GVL_IO.g_stOut.xBrakeRelease);
wTmp := F_SetBit(wTmp, 4, GVL_IO.g_stOut.xLeveling);
GVL_IO.g_awMbOut[0] := wTmp;

// DOOR_CMD
wTmp := 0;
wTmp := F_SetBit(wTmp, 0, GVL_IO.g_stOut.xDoorOpen);
wTmp := F_SetBit(wTmp, 1, GVL_IO.g_stOut.xDoorClose);
wTmp := F_SetBit(wTmp, 2, GVL_IO.g_stOut.xDoorNudge);
GVL_IO.g_awMbOut[1] := wTmp;

// Lambalar
wTmp := 0;
FOR i := 0 TO 15 DO wTmp := F_SetBit(wTmp, i, GVL_IO.g_stOut.axLampUp[i]); END_FOR
GVL_IO.g_awMbOut[2] := wTmp;

wTmp := 0;
FOR i := 0 TO 15 DO wTmp := F_SetBit(wTmp, i, GVL_IO.g_stOut.axLampDown[i]); END_FOR
GVL_IO.g_awMbOut[3] := wTmp;

wTmp := 0;
FOR i := 0 TO 15 DO wTmp := F_SetBit(wTmp, i, GVL_IO.g_stOut.axLampCar[i]); END_FOR
GVL_IO.g_awMbOut[4] := wTmp;

// STATUS_BITS
wTmp := 0;
wTmp := F_SetBit(wTmp,  0, GVL_IO.g_stOut.xMoving);
wTmp := F_SetBit(wTmp,  1, GVL_IO.g_stOut.xDoorIsOpen);
wTmp := F_SetBit(wTmp,  2, GVL_IO.g_stOut.xDoorIsClosed);
wTmp := F_SetBit(wTmp,  3, GVL_IO.g_stOut.xOverloadLamp);
wTmp := F_SetBit(wTmp,  4, GVL_IO.g_stOut.xFaultLamp);
wTmp := F_SetBit(wTmp,  5, GVL_IO.g_stOut.xFireMode);
wTmp := F_SetBit(wTmp,  6, GVL_IO.g_stOut.xInspMode);
wTmp := F_SetBit(wTmp,  7, GVL_IO.g_stOut.xOutOfService);
wTmp := F_SetBit(wTmp,  8, GVL_IO.g_stOut.xGong);
wTmp := F_SetBit(wTmp,  9, GVL_IO.g_stOut.eDirection = DIR_UP);
wTmp := F_SetBit(wTmp, 10, GVL_IO.g_stOut.eDirection = DIR_DOWN);
wTmp := F_SetBit(wTmp, 11, GVL_IO.g_stOut.xCabinLight);
wTmp := F_SetBit(wTmp, 12, GVL_IO.g_stOut.xAlarm);
GVL_IO.g_awMbOut[5] := wTmp;

GVL_IO.g_awMbOut[6]  := INT_TO_WORD(GVL_IO.g_stOut.iCurrentFloor);
GVL_IO.g_awMbOut[7]  := INT_TO_WORD(GVL_IO.g_stOut.iTargetFloor);
GVL_IO.g_awMbOut[8]  := INT_TO_WORD(GVL_IO.g_stOut.eDirection);
GVL_IO.g_awMbOut[9]  := INT_TO_WORD(GVL_IO.g_stOut.iSpeedSpMMS);
GVL_IO.g_awMbOut[10] := INT_TO_WORD(GVL_IO.g_stOut.eState);
GVL_IO.g_awMbOut[11] := INT_TO_WORD(GVL_IO.g_stOut.eFault);
GVL_IO.g_awMbOut[12] := INT_TO_WORD(GVL_IO.g_stOut.iHeartbeat);
GVL_IO.g_awMbOut[13] := INT_TO_WORD(GVL_IO.g_stOut.iDoorTimerMs);
